FUNCTION_BLOCK Station_Fault (* Basic Function Block Type *)
  (* Standard: 61499-2 *)
  (* Version 0.0, 7/14/2025, Evans_A, Schneider Electric, Template *)
  PACKAGE Main;
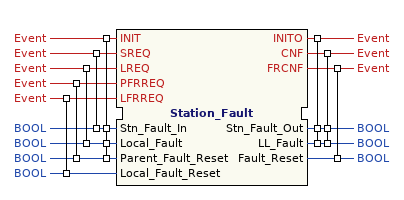
  EVENT_INPUT
    INIT WITH Stn_Fault_In, Local_Fault, Parent_Fault_Reset; (* Initialization Request *)
    SREQ WITH Stn_Fault_In; (* Normal Execution Request *)
    LREQ WITH Local_Fault;
    PFRREQ WITH Parent_Fault_Reset;
    LFRREQ WITH Local_Fault_Reset;
  END_EVENT
  EVENT_OUTPUT
    INITO WITH Stn_Fault_Out, LL_Fault; (* Initialization Confirm *)
    CNF WITH Stn_Fault_Out, LL_Fault; (* Execution Confirmation *)
    FRCNF WITH Fault_Reset;
  END_EVENT
  VAR_INPUT
    Stn_Fault_In : BOOL; (* Input event qualifier *)
    Local_Fault : BOOL;
    Parent_Fault_Reset : BOOL;
    Local_Fault_Reset : BOOL;
  END_VAR
  VAR_OUTPUT
    Stn_Fault_Out : BOOL; (* Output event qualifier *)
    LL_Fault : BOOL;
    Fault_Reset : BOOL;
  END_VAR
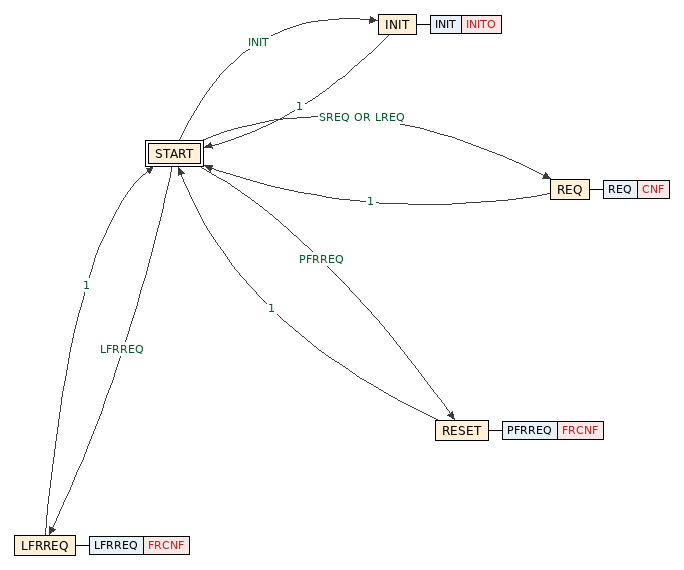
  EC_STATES
    START; (* Initial State *)
    INIT : INIT -> INITO; (* Initialization *)
    REQ : REQ -> CNF; (* Normal execution *)
    RESET : PFRREQ -> FRCNF;
    LFRREQ : LFRREQ -> FRCNF;
  END_STATES
  EC_TRANSITIONS
    START TO INIT := INIT;
    INIT TO START := 1;
    START TO REQ := SREQ OR LREQ;
    REQ TO START := 1;
    START TO RESET := PFRREQ;
    RESET TO START := 1;
    START TO LFRREQ := LFRREQ;
    LFRREQ TO START := 1;
  END_TRANSITIONS
  ALGORITHM INIT IN ST: (* Initialization algorithm *)
Stn_Fault_Out := 0;
LL_Fault := 0;
Fault_Reset := 0;
  END_ALGORITHM
  ALGORITHM REQ IN ST: (* Normally executed algorithm *)
IF Local_Fault = 1 AND Fault_Reset = 0 THEN
	LL_Fault := 1;
	Stn_Fault_Out := 1;
	Fault_Reset := 0;
ELSIF Stn_Fault_In = 1 AND Fault_Reset = 0 THEN
	LL_Fault := 0;
	Stn_Fault_Out := 1;
	Fault_Reset := 0;
ELSE
	LL_Fault := 0;
	Stn_Fault_Out := 0;
END_IF;
  END_ALGORITHM
  ALGORITHM PFRREQ IN ST:
IF Parent_Fault_Reset = 1 THEN
	Fault_Reset := 1;
	Local_Fault := 0;
	Stn_Fault_In := 0;
	Stn_Fault_Out := 0;
	LL_Fault :=0;
ELSE
	Fault_Reset := 0;
END_IF;
  END_ALGORITHM
  ALGORITHM LFRREQ IN ST:
IF Local_Fault_Reset = 1 THEN
	Fault_Reset := 1;
	Local_Fault := 0;
	LL_Fault :=0;
ELSE
	Fault_Reset := 0;
END_IF;
  END_ALGORITHM
END_FUNCTION_BLOCK
